// TIA Portal V20 export
DATA_BLOCK "instFB_HMIStatusMirror"   // DB14
TITLE = instFB_HMIStatusMirror (Phase 2.4)
VERSION : 1.1
// Phase 2.4 (C71, 2026-05-18) — instance DB for FB_HMIStatusMirror. Pure mirror FB; no statics (only VAR_TEMP for activeMode arbitration). Tiny iDB schema.
// stored: InstanceOfName FB_HMIStatusMirror, InstanceOfType FB
"FB_HMIStatusMirror"
BEGIN
END_DATA_BLOCK
